(* IEC 61131-3 sources: generating_plc_code_with_llms/Code#1/ChatGPT_3.5/third run, 21 files *)

(* ---- 14.st ---- *)
// 23.99s
// 4
FUNCTION FC1001 : BOOL
VAR_INPUT
    MeasuredValue: REAL;      // Measured value from the sensor
    SwitchingValue: REAL;     // Predetermined switching value
    HysteresisPercent: REAL;  // Switching hysteresis in percentage
END_VAR

VAR_OUTPUT
    Output: BOOL;  // Output indicating the state (ON or OFF)
END_VAR

VAR
    HysteresisValue: REAL;  // Calculated hysteresis value based on percentage
    SwitchOnThreshold: REAL; // Threshold for switching ON
    SwitchOffThreshold: REAL; // Threshold for switching OFF
END_VAR

METHOD CheckSwitching
    HysteresisValue := SwitchingValue * HysteresisPercent / 100.0;

    SwitchOnThreshold := SwitchingValue + HysteresisValue;
    SwitchOffThreshold := SwitchingValue - HysteresisValue;

    IF MeasuredValue > SwitchOnThreshold THEN
        Output := TRUE;  // Switch ON
    ELSIF MeasuredValue < SwitchOffThreshold THEN
        Output := FALSE; // Switch OFF
    END_IF
END_METHOD

END_FUNCTION

(* ---- 15.st ---- *)
// 34.7s
// 2
FUNCTION FC1002 : BOOL
VAR_INPUT
    E_A: BOOL;    // Switch for turning on/off the monitoring system
    Approach: BOOL;  // Signal from the ultrasonic sensor indicating an approach
END_VAR

VAR_OUTPUT
    P_HU: BOOL;  // Output for the acoustic warning signal
    P_AL: BOOL;  // Output for the alarm signal
    P1: BOOL;    // Output indicating the switched-on status
END_VAR

VAR
    Timer: TON := (PT := T#3s);  // Timer for tracking the duration of the approach
END_VAR

METHOD UltrasonicMonitoring
    IF E_A THEN
        P1 := TRUE;  // Monitoring system is switched on

        IF Approach THEN
            P_HU := TRUE;  // Acoustic warning signal is activated

            IF Timer(IN := TRUE).Q THEN
                // Approach duration exceeds 3 seconds, switch off warning and activate alarm
                P_HU := FALSE;
                P_AL := TRUE;
            END_IF
        ELSE
            // No approach, reset the timer and signals
            Timer(IN := FALSE);
            P_HU := FALSE;
            P_AL := FALSE;
        END_IF
    ELSE
        // Monitoring system is switched off, reset all signals
        P1 := FALSE;
        P_HU := FALSE;
        P_AL := FALSE;
        Timer(IN := FALSE);
    END_IF
END_METHOD

END_FUNCTION

(* ---- 18.st ---- *)
// 8.76s
// 2 (VAR an falscher Stelle, eigtl. 4)
FUNCTION FC1003 : REAL
VAR_INPUT
    DigitalInput: INT;  // Digital input value (0 to 255)
    IN_MIN: REAL;       // Lower limit of the original range
    IN_MAX: REAL;       // Upper limit of the original range
    OUT_MIN: REAL;      // Lower limit of the output range
    OUT_MAX: REAL;      // Upper limit of the output range
END_VAR

VAR_OUTPUT
    Temperature: REAL;  // Converted temperature value
END_VAR

METHOD MapTemperature
    // Ensure that the input is within the specified range
    IF DigitalInput < 0 THEN
        DigitalInput := 0;
    ELSIF DigitalInput > 255 THEN
        DigitalInput := 255;
    END_IF

    // Perform range mapping using linear interpolation
    Temperature := OUT_MIN + (OUT_MAX - OUT_MIN) / (IN_MAX - IN_MIN) * (DigitalInput - IN_MIN);
END_METHOD

END_FUNCTION

(* ---- 19.st ---- *)
// 18.14s
// 3
FUNCTION_BLOCK FB1005
VAR_INPUT
    START: BOOL;      // Start the measurement (connected to sensor S1)
    THICKNESS: REAL;  // Input representing the thickness of the ceramic plate
    V_MAX: REAL;      // Maximum allowed thickness
    V_MIN: REAL;      // Minimum allowed thickness
END_VAR

VAR_OUTPUT
    M_MAX: REAL;      // Largest thickness recorded during the measurement
    M_MIN: REAL;      // Smallest thickness recorded during the measurement
    P1: BOOL;         // Output for the reject light
END_VAR

VAR
    D_MAX: BOOL;      // Flag indicating if the largest thickness is outside the specified range
    D_MIN: BOOL;      // Flag indicating if the smallest thickness is outside the specified range
    ThicknessStarted: BOOL;  // Flag indicating if the thickness measurement has started
    LastThickness: REAL;     // Last recorded thickness during the measurement
END_VAR

METHOD MeasureThickness
    IF START THEN
        // Start of a new measurement cycle
        M_MAX := THICKNESS;  // Initialize largest thickness
        M_MIN := THICKNESS;  // Initialize smallest thickness
        D_MAX := FALSE;      // Initialize flags
        D_MIN := FALSE;
        ThicknessStarted := TRUE;  // Set the flag to indicate the measurement has started
    END_IF

    IF ThicknessStarted THEN
        // During the measurement cycle
        IF THICKNESS > M_MAX THEN
            M_MAX := THICKNESS;  // Update largest thickness
        END_IF

        IF THICKNESS < M_MIN THEN
            M_MIN := THICKNESS;  // Update smallest thickness
        END_IF

        LastThickness := THICKNESS;  // Record the last thickness
    END_IF

    // After the measurement cycle
    IF NOT START AND ThicknessStarted THEN
        ThicknessStarted := FALSE;  // Reset the flag to indicate the end of the measurement
        D_MAX := M_MAX > V_MAX;     // Check if the largest thickness is outside the specified range
        D_MIN := M_MIN < V_MIN;     // Check if the smallest thickness is outside the specified range
    END_IF

    // Output the reject light signal
    P1 := D_MAX OR D_MIN;
END_METHOD

END_FUNCTION_BLOCK

(* ---- 21.st ---- *)
// 49.33s
// 2
FUNCTION_BLOCK BURNER
VAR_INPUT
    IN: BOOL;              // Control input to start the burner
    OVER_TEMP: BOOL;       // Boiler thermostat protection input
    OIL_TEMP: BOOL;        // Signal indicating oil temperature
    MULTIPLE_IGNITION: BOOL;  // Allow multiple ignitions after flame failure
    STAGE2: BOOL;          // Activate second stage
    RST: BOOL;             // Reset input to restart after lockout time
END_VAR

VAR_OUTPUT
    PRE_HEAT: BOOL;        // Start fuel oil warming
    MOTOR: BOOL;           // Motor control output
    FAN: BOOL;             // Fan control output
    IGNITION: BOOL;        // Ignition control output
    OIL_VALVE: BOOL;       // Oil valve control output
    STAGE2_ACTIVATED: BOOL; // Second stage activation output
    FAIL: BOOL;            // Failure indication output
    STATUS: INT;           // Status output indicating the current state
END_VAR

VAR
    START_TIME: TIME;            // Start time of the sequence
    STAGE1_TIME: TIME := T#10s;  // Time for the first stage
    STAGE2_DELAY: TIME := T#5s;   // Delay for second stage activation
    SAFETY_TIME: TIME := T#15s;   // Safety time for flame detection
    LOCKOUT_TIME: TIME := T#300s; // Lockout time after a fault
    PRE_HEAT_TIME: TIME := T#30s; // Fuel oil warming time
    PRE_VENTILATION_TIME: TIME := T#10s; // Time for pre-ventilation
    PPR_IGNITION_TIME: TIME := T#5s;    // Time before opening the oil valve for ignition
    POST_IGNITION_TIME: TIME := T#5s;   // Time after ignition before considering the stage completed

    STAGE1_TIMER: TON := (PT := STAGE1_TIME);
    SAFETY_TIMER: TON := (PT := SAFETY_TIME);
    LOCKOUT_TIMER: TON := (PT := LOCKOUT_TIME);
    PRE_HEAT_TIMER: TON := (PT := PRE_HEAT_TIME);
    PRE_VENTILATION_TIMER: TON := (PT := PRE_VENTILATION_TIME);
    PPR_IGNITION_TIMER: TON := (PT := PPR_IGNITION_TIME);
    POST_IGNITION_TIMER: TON := (PT := POST_IGNITION_TIME);
    STAGE2_DELAY_TIMER: TON := (PT := STAGE2_DELAY);
END_VAR

METHOD BurnerControl
    // Status initialization
    STATUS := 110; // Wait for Start signal (Standby)
    FAIL := FALSE;

    IF RST AND LOCKOUT_TIMER.Q THEN
        // Reset after the lockout time has passed
        LOCKOUT_TIMER(IN := FALSE);
    END_IF

    // Burner operation control
    CASE STATUS OF
        110: // Wait for Start signal (Standby)
            IF IN AND NOT OVER_TEMP THEN
                STATUS := 111; // Startup sequence is executed
                START_TIME := TIME();
                PRE_HEAT := TRUE;
            END_IF
        111: // Startup sequence is executed
            IF PRE_HEAT_TIMER.Q THEN
                PRE_HEAT := FALSE;
                MOTOR := TRUE; // Start the motor
                FAN := TRUE;   // Start the fan
                STAGE1_TIMER(IN := TRUE);
            END_IF

            IF STAGE1_TIMER.Q THEN
                // First stage completed
                IGNITION := TRUE; // Start ignition
                PPR_IGNITION_TIMER(IN := TRUE);
                STATUS := 112; // Burner runs on stage 1
            END_IF
        112: // Burner runs on stage 1
            IF MULTIPLE_IGNITION AND PPR_IGNITION_TIMER.Q THEN
                // Ignition failed, start another ignition attempt
                IGNITION := TRUE;
                PPR_IGNITION_TIMER(IN := TRUE);
            END_IF

            IF PPR_IGNITION_TIMER.Q THEN
                // Ignition completed, open the oil valve
                IGNITION := FALSE;
                OIL_VALVE := TRUE;
                POST_IGNITION_TIMER(IN := TRUE);
            END_IF

            IF POST_IGNITION_TIMER.Q THEN
                // First stage completed
                STATUS := 113; // Burner runs on stage 2
                STAGE2_ACTIVATED := TRUE;
                STAGE2_DELAY_TIMER(IN := TRUE);
            END_IF
        113: // Burner runs on stage 2
            IF STAGE2_DELAY_TIMER.Q THEN
                // Second stage activated
                STAGE2_ACTIVATED := STAGE2;
            END_IF

            // Check for flame failure
            IF SAFETY_TIMER.Q AND (IGNITION OR OIL_VALVE) THEN
                FAIL := TRUE; // Flame failure
                STATUS := 5;   // Fame stops in operation
            END_IF
    END_CASE

    // Check for lockout conditions
    IF OVER_TEMP THEN
        STATUS := 9;  // Boiler overheating contact has tripped
    END_IF

    // Update status and initiate lockout if needed
    IF STATUS <> 9 AND (FAIL OR (RST AND NOT LOCKOUT_TIMER.Q)) THEN
        STATUS := 110; // Wait for Start signal (Standby)
        LOCKOUT_TIMER(IN := TRUE); // Initiate lockout
    END_IF
END_METHOD

END_FUNCTION_BLOCK

(* ---- 1.st ---- *)
//6.87s
//2
PROGRAM AlarmControl
VAR
    xAlarm1: BOOL := FALSE;
    xAlarm2: BOOL := FALSE;
    xAllOn: BOOL := FALSE;
    xAllOff: BOOL := FALSE;
END_VAR

METHOD TurnAllAlarmsOff : BOOL
    xAlarm1 := FALSE;
    xAlarm2 := FALSE;
    RETURN TRUE;
END_METHOD

METHOD TurnAllAlarmsOn : BOOL
    xAlarm1 := TRUE;
    xAlarm2 := TRUE;
    RETURN TRUE;
END_METHOD

IF xAllOn THEN
    TurnAllAlarmsOn();
    xAllOn := FALSE;  // Reset the signal
ELSIF xAllOff THEN
    TurnAllAlarmsOff();
    xAllOff := FALSE; // Reset the signal
END_IF

(* ---- 10.st ---- *)
//5.18s
//2
PROGRAM SigmoidFunction
VAR_INPUT
    x: REAL;  // Input value for the sigmoid function
END_VAR

VAR_OUTPUT
    sigmoidResult: REAL;  // Output value of the sigmoid function
END_VAR

METHOD CalculateSigmoid
    sigmoidResult := 1.0 / (1.0 + EXP(-x));
END_METHOD

END_PROGRAM

(* ---- 11.st ---- *)
//6.88s
//2
PROGRAM SignFunction
VAR_INPUT
    x: REAL;  // Input value for the sign function
END_VAR

VAR_OUTPUT
    signResult: INT;  // Output value of the sign function (-1, 0, or 1)
END_VAR

METHOD CalculateSign
    IF x < 0.0 THEN
        signResult := -1;
    ELSIF x > 0.0 THEN
        signResult := 1;
    ELSE
        signResult := 0;
    END_IF
END_METHOD

END_PROGRAM

(* ---- 12.st ---- *)
//6.35s
//2
PROGRAM SignFunction
VAR_INPUT
    x: REAL;  // Input value for the sign function
END_VAR

VAR_OUTPUT
    signResult: INT;  // Output value of the sign function (-1, 0, or 1)
END_VAR

METHOD CalculateSign
    IF x < 0.0 THEN
        signResult := -1; // Negative value
    ELSIF x > 0.0 THEN
        signResult := 1;  // Positive value
    ELSE
        signResult := 0;  // Zero
    END_IF
END_METHOD

END_PROGRAM

(* ---- 13.st ---- *)
//8.89s
//2; wenn VAR richtig, immernoch falsch
PROGRAM NumberSearch
VAR
    NumberList: ARRAY[1..100] OF INT;  // List of 100 random numbers
    FoundTen: BOOL := FALSE;  // Flag to indicate if the number 10 is found
    i: INT := 1;  // Loop variable
END_VAR

METHOD SearchNumber
    REPEAT
        IF NumberList[i] = 10 THEN
            FoundTen := TRUE;  // Number 10 is found, abort the search
            EXIT;
        END_IF
        i := i + 1;  // Move to the next number in the list

        IF i > 100 THEN
            EXIT;  // All elements have been checked, abort the search
        END_IF
    UNTIL FoundTen OR i > 100;
END_METHOD

END_PROGRAM

(* ---- 16.st ---- *)
//11.85s
//2
PROGRAM TrafficLightControl
VAR
    North_green: BOOL := FALSE;
    North_yellow: BOOL := FALSE;
    North_red: BOOL := FALSE;
    East_green: BOOL := FALSE;
    East_yellow: BOOL := FALSE;
    East_red: BOOL := FALSE;
    TrafficLightTimer: TON := (PT := T#10000ms);
END_VAR

METHOD ControlTrafficLights
    IF NOT TrafficLightTimer.IN THEN
        // Timer has not started yet, initialize the lights
        North_green := TRUE;
        East_red := TRUE;
    ELSE
        IF TrafficLightTimer.Q THEN
            // Timer has completed one cycle, reset it
            TrafficLightTimer(IN := FALSE);
        ELSE
            // Traffic light sequence within one cycle
            IF TrafficLightTimer.ET > T#0ms AND TrafficLightTimer.ET <= T#5000ms THEN
                North_green := TRUE;
                East_red := TRUE;
                North_yellow := FALSE;
                East_yellow := FALSE;
                North_red := FALSE;
            ELSIF TrafficLightTimer.ET > T#5000ms AND TrafficLightTimer.ET <= T#5500ms THEN
                North_green := FALSE;
                North_yellow := TRUE;
                North_red := FALSE;
            ELSIF TrafficLightTimer.ET > T#5500ms AND TrafficLightTimer.ET <= T#9500ms THEN
                North_green := FALSE;
                East_red := FALSE;
                North_yellow := FALSE;
                East_yellow := FALSE;
                North_red := TRUE;
                East_green := TRUE;
            ELSIF TrafficLightTimer.ET > T#9500ms AND TrafficLightTimer.ET <= T#10000ms THEN
                East_green := FALSE;
                East_yellow := TRUE;
                East_red := FALSE;
            END_IF
        END_IF
    END_IF
END_METHOD

END_PROGRAM

(* ---- 17.st ---- *)
//10.61s
//2 Var an falscher Stelle, sonst 4
PROGRAM WeatherStation
VAR_INPUT
    Temperature: INT;  // Input temperature in degrees Celsius (0 - 100)
    Humidity: INT;     // Input humidity in percentage (0 - 100)
END_VAR

VAR_OUTPUT
    DisplayText: STRING := '';  // Output text for display
END_VAR

METHOD DisplayWeatherStatus
    IF Temperature < 18 THEN
        DisplayText := 'Cold';
    ELSIF Temperature >= 18 AND Temperature <= 25 AND Humidity >= 40 AND Humidity <= 75 THEN
        DisplayText := 'Opt';
    ELSIF Temperature > 25 THEN
        DisplayText := 'Hot';
    ELSE
        DisplayText := 'Temp. OK';
    END_IF
END_METHOD

END_PROGRAM

(* ---- 2.st ---- *)
//6.82s
//4
PROGRAM BinomialCoefficient
VAR_INPUT
    n: UINT; // Total number of items
    k: UINT; // Number of items to choose
END_VAR

VAR_OUTPUT
    binomialCoeff: UINT; // Binomial coefficient result
END_VAR

VAR
    i: UINT;
    j: UINT;
    result: UINT;
END_VAR

METHOD CalculateBinomialCoeff
    IF k > n THEN
        binomialCoeff := 0; // Invalid input, k cannot be greater than n
    ELSE
        result := 1;
        FOR i := 1 TO k DO
            result := result * (n - i + 1) / i;
        END_FOR
        binomialCoeff := result;
    END_IF
END_METHOD

END_PROGRAM

(* ---- 20.st ---- *)
// 17.82s
// 3
PROGRAM InterlockProgram
VAR_INPUT
    I1: BOOL;  // Input to switch Q1
    I2: BOOL;  // Input to switch Q2
END_VAR

VAR_OUTPUT
    Q1: BOOL;  // Output Q1
    Q2: BOOL;  // Output Q2
END_VAR

VAR
    TimerQ1: TON := (PT := T#1s);  // Timer for Q1
    TimerQ2: TON := (PT := T#1s);  // Timer for Q2
    TL: TIME := T#500ms;           // Dead time between Q1 and Q2
    LastQ1State: BOOL := FALSE;    // Last state of Q1
    LastQ2State: BOOL := FALSE;    // Last state of Q2
END_VAR

METHOD InterlockLogic
    // Update timers
    TimerQ1(IN := I1);
    TimerQ2(IN := I2);

    // Determine the next state of Q1
    IF I1 AND NOT Q2 AND TimerQ2.Q THEN
        Q1 := TRUE;
        LastQ1State := TRUE;
    ELSIF NOT I1 THEN
        Q1 := FALSE;
        TimerQ1(IN := FALSE);  // Reset the timer if I1 is OFF
    END_IF

    // Determine the next state of Q2
    IF I2 AND NOT Q1 AND TimerQ1.Q THEN
        Q2 := TRUE;
        LastQ2State := TRUE;
    ELSIF NOT I2 THEN
        Q2 := FALSE;
        TimerQ2(IN := FALSE);  // Reset the timer if I2 is OFF
    END_IF

    // Check for mutual locking
    IF LastQ1State AND TimerQ2.ET < TL THEN
        Q1 := FALSE;
    END_IF

    IF LastQ2State AND TimerQ1.ET < TL THEN
        Q2 := FALSE;
    END_IF

    // Update last states
    LastQ1State := Q1;
    LastQ2State := Q2;
END_METHOD

END_PROGRAM

(* ---- 3.st ---- *)
//7.84
//3
PROGRAM FibonacciCalculation
VAR_INPUT
    n: INT; // The position of the Fibonacci number to calculate
END_VAR

VAR_OUTPUT
    fibonacciNumber: INT; // The calculated Fibonacci number
END_VAR

VAR
    i: INT;
    fib1: INT := 0; // Initialize the first Fibonacci number
    fib2: INT := 1; // Initialize the second Fibonacci number
END_VAR

METHOD CalculateFibonacci
    IF n <= 0 THEN
        fibonacciNumber := 0; // Fibonacci number at position 0 or negative positions
    ELSIF n = 1 THEN
        fibonacciNumber := 1; // Fibonacci number at position 1
    ELSE
        FOR i := 2 TO n DO
            fibonacciNumber := fib1 + fib2;
            fib1 := fib2;
            fib2 := fibonacciNumber;
        END_FOR
    END_IF
END_METHOD

END_PROGRAM

(* ---- 4.st ---- *)
//10.25s
//2
PROGRAM FillLevelCheck
VAR_INPUT
    analogValue: INT := 0 TO 32767; // Input analog value (0 - 32767)
END_VAR

VAR_OUTPUT
    lowLevel: BOOL := FALSE;  // Output for low fill level
    okLevel: BOOL := FALSE;   // Output for ok fill level
    highLevel: BOOL := FALSE; // Output for high fill level
    warningHorn: BOOL := FALSE; // Output for warning horn
END_VAR

VAR
    fillLevelPercentage: INT := 0 TO 100; // Internal variable for fill level in percentage
END_VAR

CASE fillLevelPercentage OF
    (0 TO 1):   // Below 1%
        lowLevel := FALSE;
        okLevel := FALSE;
        highLevel := FALSE;
        warningHorn := TRUE;
    (2 TO 70):  // 2% to 70%
        lowLevel := FALSE;
        okLevel := TRUE;
        highLevel := FALSE;
        warningHorn := FALSE;
    (71 TO 100): // 71% to 100%
        lowLevel := FALSE;
        okLevel := FALSE;
        highLevel := TRUE;
        warningHorn := FALSE;
    ELSE        // Any other values
        lowLevel := TRUE;
        okLevel := FALSE;
        highLevel := FALSE;
        warningHorn := FALSE;
END_CASE

END_PROGRAM

(* ---- 5.st ---- *)
//10.7s
//2
PROGRAM GateController
VAR_INPUT
    Start_Loop: BOOL;        // Input to start the gate controller
    Gate_Open: BOOL;         // Input indicating whether the gate is open
    App_Presence: BOOL;      // Input indicating the presence of the app
    Car_Presence: BOOL;      // Input indicating the presence of the car
    Auth_String: STRING;     // Input authentication string
END_VAR

VAR_OUTPUT
    Gate_Control: BOOL;      // Output to control the gate (TRUE to open, FALSE to close)
END_VAR

VAR
    One_Hour_Timer: TON;     // One-hour timer
    Timer_Done: BOOL;        // Timer done flag
    Auth_Matched: BOOL;      // Authentication string match flag
    My_Defined_Str: STRING := "your_defined_string"; // Replace with your actual authentication string
END_VAR

METHOD OpenGate
    Gate_Control := TRUE;
END_METHOD

METHOD CloseGate
    Gate_Control := FALSE;
END_METHOD

IF Start_Loop THEN
    One_Hour_Timer(IN := FALSE);
    Timer_Done := FALSE;
    Auth_Matched := FALSE;
ELSE
    One_Hour_Timer(IN := TRUE, PT := T#1H);  // Start the 1-hour timer when Start_Loop is FALSE
    IF One_Hour_Timer.Q THEN
        Timer_Done := TRUE;  // Timer has timed out
        IF Gate_Open THEN
            CloseGate();  // Close the gate if it's still open
        END_IF
    END_IF
    IF (App_Presence OR Car_Presence) AND Auth_String = My_Defined_Str THEN
        Auth_Matched := TRUE;  // Authentication string matches, and either the app or car is present
        OpenGate();  // Open the gate
    END_IF
END_IF

END_PROGRAM

(* ---- 6.st ---- *)
//16.58s
//2
PROGRAM CraneLiftSystem
VAR
    doConvTop: BOOL := FALSE;     // Conveyor belt for top
    doConvBottom: BOOL := FALSE;  // Conveyor belt for bottom
    diConvTop: BOOL := FALSE;     // Light barrier for top conveyor
    diConvBottom: BOOL := FALSE;  // Light barrier for bottom conveyor
    doLiftTop: BOOL := FALSE;     // Lift control for top position
    doLiftBottom: BOOL := FALSE;  // Lift control for bottom position
    diLiftTop: BOOL := FALSE;     // Lift position for top
    diLiftBottom: BOOL := FALSE;  // Lift position for bottom
    doConvLift: BOOL := FALSE;    // Conveyor belt on the lift
    diBoxLift: BOOL := FALSE;     // Crate at the lift
    doLiftUnload: BOOL := FALSE;  // Lift control for unloading position
    diLiftUnload: BOOL := FALSE;  // Lift position for unloading
END_VAR

METHOD RequestLift
    IF diConvTop AND NOT doLiftTop THEN
        doConvTop := FALSE;    // Stop the top conveyor
        doLiftTop := TRUE;     // Move the lift to the top position
    ELSIF diConvBottom AND NOT doLiftBottom THEN
        doConvBottom := FALSE; // Stop the bottom conveyor
        doLiftBottom := TRUE;  // Move the lift to the bottom position
    END_IF
END_METHOD

METHOD MoveLift
    IF doLiftTop AND diLiftTop THEN
        doConvLift := TRUE;    // Turn on the lift conveyor
        IF diBoxLift THEN
            doLiftTop := FALSE; // Move the lift to unloading position
            doLiftUnload := TRUE;
        END_IF
    ELSIF doLiftBottom AND diLiftBottom THEN
        doConvLift := TRUE;    // Turn on the lift conveyor
        IF diBoxLift THEN
            doLiftBottom := FALSE;  // Move the lift to unloading position
            doLiftUnload := TRUE;
        END_IF
    END_IF
END_METHOD

METHOD UnloadLift
    IF doLiftUnload AND diLiftUnload THEN
        doConvLift := FALSE; // Turn off the lift conveyor
        doLiftUnload := FALSE; // Reset the lift control for unloading position
        // Place code here to convey the crate from the lift to the unloading conveyor
    END_IF
END_METHOD

END_PROGRAM

(* ---- 7.st ---- *)
//9.64
//2 wenn Var richtig, dann 4
PROGRAM CraneControl
VAR_INPUT
    LoadReceptor: ARRAY[1..5] OF INT := [0, 0, 0, 0, 0]; // Input load values from 0 to 32767
END_VAR

VAR_OUTPUT
    TotalLoad: INT := 0;  // Output for total load
    AverageLoad: INT := 0;  // Output for average load
END_VAR

VAR
    NumLoadReceptors: INT := 5;  // Number of load receptors
    i: INT;  // Loop variable
    LoadSum: INT := 0;  // Total load accumulator
END_VAR

METHOD CalculateLoad
    LoadSum := 0;

    FOR i := 1 TO NumLoadReceptors DO
        LoadSum := LoadSum + LoadReceptor[i];
    END_FOR

    IF NumLoadReceptors > 0 THEN
        AverageLoad := LoadSum / NumLoadReceptors;
    ELSE
        AverageLoad := 0; // Avoid division by zero
    END_IF

    TotalLoad := LoadSum;
END_METHOD

END_PROGRAM

(* ---- 8.st ---- *)
//11.22s
//2 eigentlich ausführbar, aber VAR an der falschen Stelle
PROGRAM LambertWApproximation
VAR_INPUT
    x: REAL; // Input value for the Lambert W function
END_VAR

VAR_OUTPUT
    LambertW: REAL; // Output value of the Lambert W function
END_VAR

VAR
    maxIterations: INT := 100;  // Maximum number of iterations
    tolerance: REAL := 1.0E-6; // Tolerance for convergence
    y, yPrev: REAL;
    i: INT;
END_VAR

METHOD LambertWApproximate
    IF x < -1.0 / exp(1.0) THEN
        // Handle the case where x is outside the domain of Lambert W
        LambertW := 0.0;
    ELSE
        // Initialize the approximate value
        y := MAX(x, -1.0 + tolerance);

        FOR i := 1 TO maxIterations DO
            yPrev := y;
            y := y - ((y * exp(y) - x) / (exp(y) + y * exp(y)));

            IF ABS(y - yPrev) < tolerance THEN
                // Convergence achieved
                LambertW := y;
                RETURN;
            END_IF
        END_FOR

        // If the loop completes without convergence, Lambert W is not valid
        LambertW := 0.0;
    END_IF
END_METHOD

END_PROGRAM

(* ---- 9.st ---- *)
//7.42s
//2
PROGRAM LeapYearCheck
VAR_INPUT
    YEAR: INT; // Input year to check
END_VAR

VAR_OUTPUT
    IsLeapYear: BOOL; // Output indicating whether the year is a leap year
END_VAR

METHOD CheckLeapYear
    IF ((YEAR MOD 4 = 0) AND (YEAR MOD 100 <> 0)) OR (YEAR MOD 400 = 0) THEN
        IsLeapYear := TRUE; // It's a leap year
    ELSE
        IsLeapYear := FALSE; // It's not a leap year
    END_IF
END_METHOD

END_PROGRAM
